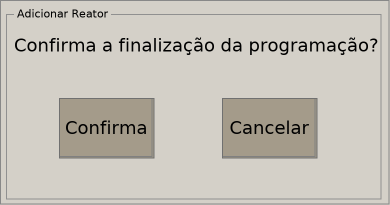
VISUALIZATION FinalizaProg  // 390x205
VAR_IN_OUT
	bReator: BOOL;
	iOFnumber: INT;
	iSrlNumber: INT;
	
	
	
END_VAR
    GroupBox (6,6 375x193), "Adicionar Reator"
        Button (53,92 95x60), "Confirma"
            OnMouseClick: CloseDialog Dialog=FinalizaProg, Result=OK, NumpadKeypadSet=True
            OnMouseClick: execute {
                IF gvl.actEst = 0 THEN
                	Rotina019.status:= 45;
                	Rotina019_Manual.status:= 45;
                ELSIF gvl.actEst = 1 THEN
                	Rotina020.status:= 45;
                	Rotina020_Manual.status:=45;
                ELSIF gvl.actEst = 2 THEN
                	Rotina021.status:= 45;
                	Rotina021_Manual.status:= 45;
                END_IF
            }
        Button (216,92 95x60), "Cancelar"
            OnMouseClick: CloseDialog Dialog=FinalizaProg, Result=Cancel, NumpadKeypadSet=True
        Label (5,27 381x63), "Confirma a finalização da programação?"
END_VISUALIZATION

(* stored: Version 1.1.0.1, ProductVersion 3.1.4024.12
   Visu FinalizaProg: Id {662489c4-7e06-498a-9a35-ab20acdb3a29} *)
